(*
A broadcastable wrapper for a `BOOL` value. 
*)
FUNCTION_BLOCK BoolArg IMPLEMENTS I_BoolArg
VAR
	_val			: BOOL;
	_bMut			: BOOL := FALSE;
END_VAR

(*
Enables external modification of the internal value.
*)
METHOD AllowMut
_bMut := TRUE;
END_METHOD

(*
Disables external modification of the internal value.
*)
METHOD BlockMut
_bMut := FALSE;
END_METHOD

//FB_Init is always available implicitly and it is used primarily for initialization.
//The return value is not evaluated. For a specific influence, you can also declare the
//methods explicitly and provide additional code there with the standard initialization
//code. You can evaluate the return value.
{attribute 'hide'}
METHOD FB_Init: BOOL
VAR_INPUT
    bInitRetains: BOOL; // TRUE: the retain variables are initialized (reset warm / reset cold)
    bInCopyCode: BOOL;  // TRUE: the instance will be copied to the copy code afterward (online change)   

	initVal		: BOOL;
END_VAR
_val := initVal;
END_METHOD

(*
Reads the internal value.
*)
PROPERTY Get : BOOL
GET
Get := _val;
END_GET
END_PROPERTY

(*
Returns TRUE if the value is mutable.
*)
PROPERTY IsMut : BOOL
GET
IsMut := _bMut;
END_GET
END_PROPERTY

(*
Directly modifies the internal value, bypassing any mutability restrictions.
*)
METHOD OpSet : I_Arg
VAR_INPUT
	newVal		: BOOL;
END_VAR
_val := newVal;
OpSet := THIS^;
END_METHOD

(*
Modifies the internal value.  
Returns:
- `Ok` - Upon successful modification.
- `Error` - If mutability is disabled.
*)
METHOD Set : Result
VAR_INPUT
	newVal		: BOOL;
END_VAR
IF _bMut THEN
	_val := newVal;
	Set := Ok;
ELSE
	Set := Error;
END_IF
END_METHOD

END_FUNCTION_BLOCK

(* stored: Version 1.1.0.1
   POU BoolArg: Id {e27e2f24-10ad-4112-bcdb-e1d34b1a5e15}, SpecialFunc None
   Method AllowMut: Id {4f24b0df-f054-4394-8fe0-e220d5913655}
   Method BlockMut: Id {5208fcfc-5d8b-46e0-8ceb-90e6e73bcbfb}
   Method FB_Init: Id {7c178ce6-db6f-4695-91ea-604be15c984e}
   Property Get: Id {6ed6bcd8-cacc-489e-b1d3-a9fb999002c0}
   Get Get: Id {c4b33677-e84c-45d8-8f95-32db6a3146a4}
   Property IsMut: Id {099e7873-cad3-4196-9c99-cd99bbe92bf2}
   Get Get: Id {84380cb3-20b1-4148-a377-a167c62be6ec}
   Method OpSet: Id {2d73b277-04bf-4aa2-be85-20bda0268174}
   Method Set: Id {45e10697-aae4-4067-adec-6d3af11582dd} *)
